// TIA Portal V20 export
DATA_BLOCK "PM1"   // DB273
// stored: MemoryReserve 100
   VAR
      "STACK #1 NG CLAMP MOVER CLOSE" : Bool;
      "STACK #1 NG CLAMP MOVER OPEN" : Bool;
      "STACK #1 NG CLAMP RIGHT CLOSE" : Bool;
      "STACK #1 NG CLAMP RIGHT OPEN" : Bool;
      "STACK #1 NG CLAMP LEFT OPEN" : Bool;
      "STACK #1 NG CLAMP LEFT CLOSE" : Bool;
      "STAKC #1 NG CLAMP Z-AXIS UP" : Bool;
      "STAKC #1 NG CLAMP Z-AXIS DOWN" : Bool;
      "STAKC #1 NG CLAMP MOVER FORWARD" : Bool;
      "STAKC #1 NG CLAMP MOVER BACKWARD" : Bool;
      "STACK #1 NG BOX LIFT UP" : Bool;
      "STACK #1 NG BOX LIFT DOWN" : Bool;
      "STACK #1 NG BOX LOCK UP" : Bool;
      "STACK #1 NG BOX LOCK DOWN" : Bool;
      "JR OUT P&P#1 CLAMP CLOSE" : Bool;
      "JR OUT P&P#1 CLAMP OPEN" : Bool;
   END_VAR
BEGIN
END_DATA_BLOCK
